PROGRAM Set_Strand_Calib
VAR PERSISTENT
	
	Set_Calibration_Factor : BOOL;
	Actual_Measured_Diameter : REAL;
END_VAR

IF Set_Calibration_Factor THEN
	GVL_Vision.Calibration_Factor := Diameter_Algo.StrandWidth / Actual_Measured_Diameter; //Calcualted pixels / actual strand diameter;
END_IF

END_PROGRAM

(* stored: Version 1.1.0.1, ProductVersion 3.1.4024.12
   POU Set_Strand_Calib: Id {1d612d15-6097-418a-a1a0-4c718f532339}, SpecialFunc None *)
